// TIA Portal V17 export
// export: Created 2022-04-06T07:28:40.7183202Z, ExportSetting WithDefaults, DisplayName Totally Integrated Automation Portal, DisplayVersion V17, DisplayName TIA Portal Openness, DisplayVersion V17, DisplayName TIA Portal Version Control Interface, DisplayVersion V17, DisplayName TIA Portal Test Suite Advanced, DisplayVersion V17, DisplayName SINAMICS Startdrive Advanced, DisplayVersion V17, DisplayName SINAMICS Startdrive G130, G150, S120, S150, SINAMICS MV, S210, DisplayVersion V17, DisplayName SINAMICS Startdrive G110M, G120, G120C, G120D, G120P, G115D, DisplayVersion V17, DisplayName STEP 7 Professional, DisplayVersion V17, DisplayName STEP 7 Safety, DisplayVersion V17, DisplayName WinCC Advanced / Unified PC, DisplayVersion V17
TYPE "LDrvSafe_typeSinaSTlg30Control"
TITLE = LDrvSafe_typeSinaSTlg30Control
// Failsafe user-defined data type for PROFIsafe telegram 30 to control the Safety Integrated Functions of SINAMICS S
// stored: IsFailsafeCompliant true
   STRUCT
      STO { ExternalWritable := 'False'} : Bool;   // Safety Function Safe Torque Off
      SS1 { ExternalWritable := 'False'} : Bool;   // Safety Function Safe Stop 1
      SS2 { ExternalWritable := 'False'} : Bool;   // Safety Function Safe Stop 2
      SOS { ExternalWritable := 'False'} : Bool;   // Safety Function Safe Operating Stop
      SLS { ExternalWritable := 'False'} : Bool;   // Safety Function Safely-limited Speed
      reserved1 { ExternalWritable := 'False'} : Bool;   // Reserve bit 1
      SLP { ExternalWritable := 'False'} : Bool;   // Safety Function Safely-limited Position
      internalEventAcknowledge { ExternalWritable := 'False'} : Bool;   // Acknowledge Safety errors in the drive
      SLA { ExternalWritable := 'False'} : Bool;   // Safety Function Safely-limited Acceleration
      selectSLSbit0 { ExternalWritable := 'False'} : Bool;   // Select one of the the four SLS limits; operates together with bit 1
      selectSLSbit1 { ExternalWritable := 'False'} : Bool;   // Select one of the the four SLS limits; operates together with bit 0
      reserved3 { ExternalWritable := 'False'} : Bool;   // Reserve bit 3
      SDIpositive { ExternalWritable := 'False'} : Bool;   // Safety Function Safe Direction (positive direction)
      SDInegative { ExternalWritable := 'False'} : Bool;   // Safety Function Safe Direction (negative direction)
      reserved4 { ExternalWritable := 'False'} : Bool;   // Reserve bit 4
      reserved5 { ExternalWritable := 'False'} : Bool;   // Reserve bit 5
   END_STRUCT;
END_TYPE
